FUNCTION_BLOCK FB_TriLogic (* Logique de tri - BLOCK seulement si couleur differente *)
  (* Standard: 61499-2 *)
  (* Version 2.0, 20/01/2026, Claude, Schneider Electric, Block seulement si changement de couleur *)
  PACKAGE Main;
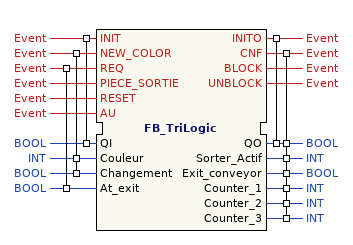
  EVENT_INPUT
    INIT WITH QI; (* Initialization Request *)
    NEW_COLOR WITH Couleur, Changement; (* Nouvelle couleur detectee *)
    REQ WITH At_exit; (* Cyclic update *)
    PIECE_SORTIE; (* Piece a quitte le systeme (front descendant At_exit) *)
    RESET; (* Reset compteurs *)
    AU; (* Arret urgence *)
  END_EVENT
  EVENT_OUTPUT
    INITO WITH QO; (* Initialization Confirm *)
    CNF WITH QO, Sorter_Actif, Exit_conveyor, Counter_1, Counter_2, Counter_3; (* Execution Confirmation *)
    BLOCK; (* Bloquer entree (couleur differente) *)
    UNBLOCK; (* Debloquer entree *)
  END_EVENT
  VAR_INPUT
    QI : BOOL; (* Input event qualifier *)
    Couleur : INT; (* 1=Bleu, 2=Vert, 3=Gris *)
    Changement : BOOL; (* TRUE si couleur differente *)
    At_exit : BOOL; (* Capteur sortie *)
  END_VAR
  VAR_OUTPUT
    QO : BOOL; (* Output event qualifier *)
    Sorter_Actif : INT; (* Sorter actif (1-3) *)
    Exit_conveyor : BOOL; (* Convoyeur sortie actif *)
    Counter_1 : INT; (* Compteur bleu *)
    Counter_2 : INT; (* Compteur vert *)
    Counter_3 : INT; (* Compteur gris *)
  END_VAR
  VAR
    Couleur_EnCours : INT; (* Couleur piece en cours de tri *)
    Couleur_Suivante : INT; (* Couleur piece suivante (si differente) *)
    Is_Blocked : BOOL; (* TRUE si entree bloquee *)
  END_VAR
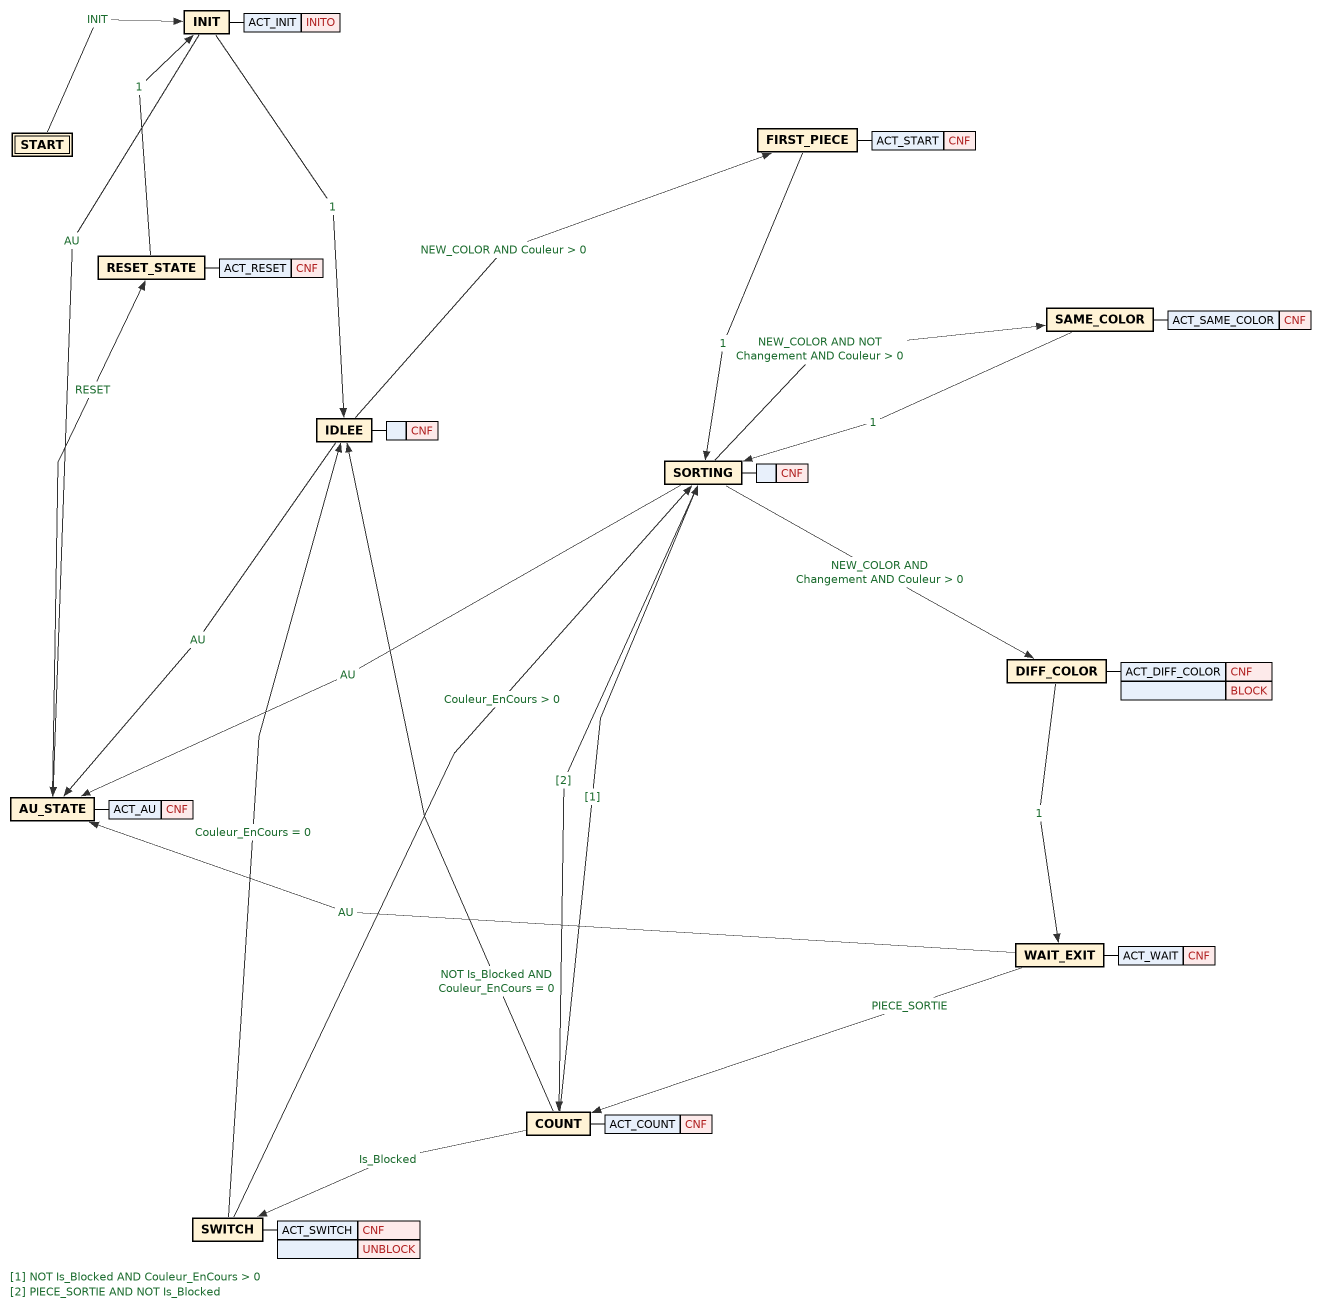
  EC_STATES
    START; (* Initial State *)
    INIT : ACT_INIT -> INITO; (* Initialization *)
    IDLEE : -> CNF; (* En attente - pas de piece *)
    FIRST_PIECE : ACT_START -> CNF; (* Premiere piece - activer sorter *)
    SORTING : -> CNF; (* Tri en cours *)
    SAME_COLOR : ACT_SAME_COLOR -> CNF; (* Meme couleur - pas de blocage *)
    DIFF_COLOR : ACT_DIFF_COLOR -> CNF, -> BLOCK; (* Couleur differente - BLOCK *)
    WAIT_EXIT : ACT_WAIT -> CNF; (* Attendre sortie piece *)
    COUNT : ACT_COUNT -> CNF; (* Piece sortie - compter *)
    SWITCH : ACT_SWITCH -> CNF, -> UNBLOCK; (* Changer sorter - UNBLOCK *)
    AU_STATE : ACT_AU -> CNF; (* Arret urgence *)
    RESET_STATE : ACT_RESET -> CNF; (* Reset *)
  END_STATES
  EC_TRANSITIONS
    START TO INIT := INIT;
    INIT TO IDLEE := 1;
    IDLEE TO FIRST_PIECE := NEW_COLOR AND Couleur > 0;
    FIRST_PIECE TO SORTING := 1;
    SORTING TO SAME_COLOR := NEW_COLOR AND NOT Changement AND Couleur > 0;
    SORTING TO DIFF_COLOR := NEW_COLOR AND Changement AND Couleur > 0;
    SAME_COLOR TO SORTING := 1;
    DIFF_COLOR TO WAIT_EXIT := 1;
    WAIT_EXIT TO COUNT := PIECE_SORTIE;
    SORTING TO COUNT := PIECE_SORTIE AND NOT Is_Blocked;
    COUNT TO SWITCH := Is_Blocked;
    COUNT TO SORTING := NOT Is_Blocked AND Couleur_EnCours > 0;
    COUNT TO IDLEE := NOT Is_Blocked AND Couleur_EnCours = 0;
    SWITCH TO SORTING := Couleur_EnCours > 0;
    SWITCH TO IDLEE := Couleur_EnCours = 0;
    IDLEE TO AU_STATE := AU;
    SORTING TO AU_STATE := AU;
    WAIT_EXIT TO AU_STATE := AU;
    AU_STATE TO RESET_STATE := RESET;
    RESET_STATE TO INIT := 1;
    INIT TO AU_STATE := AU;
  END_TRANSITIONS
  ALGORITHM ACT_INIT IN ST: (* Initialization *)
QO := TRUE;
Sorter_Actif := 0;
Exit_conveyor := FALSE;
Couleur_EnCours := 0;
Couleur_Suivante := 0;
Is_Blocked := FALSE;
Counter_1 := 0;
Counter_2 := 0;
Counter_3 := 0;
  END_ALGORITHM
  ALGORITHM ACT_START IN ST: (* Premiere piece - activer sorter *)
(* Premiere piece detectee - activer le sorter *)
Couleur_EnCours := Couleur;
Sorter_Actif := Couleur;
Exit_conveyor := TRUE;
Is_Blocked := FALSE;
  END_ALGORITHM
  ALGORITHM ACT_SAME_COLOR IN ST: (* Meme couleur - continuer sans bloquer *)
(* Meme couleur que precedente - pas de blocage *)
(* Le sorter est deja bon, on continue *)
Exit_conveyor := TRUE;
  END_ALGORITHM
  ALGORITHM ACT_DIFF_COLOR IN ST: (* Couleur differente - bloquer et memoriser *)
(* Couleur DIFFERENTE - bloquer l'entree et memoriser *)
Couleur_Suivante := Couleur;
Is_Blocked := TRUE;
(* IMPORTANT: garder le sorter actuel jusqu'a ce que la piece sorte *)
Exit_conveyor := TRUE;
  END_ALGORITHM
  ALGORITHM ACT_WAIT IN ST: (* Attendre sortie piece *)
(* Attendre que la piece en cours sorte *)
(* Garder le sorter actuel actif *)
Sorter_Actif := Couleur_EnCours;
Exit_conveyor := TRUE;
  END_ALGORITHM
  ALGORITHM ACT_COUNT IN ST: (* Compter la piece sortie *)
(* Piece sortie - incrementer compteur *)
IF Couleur_EnCours = 1 THEN
    Counter_1 := Counter_1 + 1;
ELSIF Couleur_EnCours = 2 THEN
    Counter_2 := Counter_2 + 1;
ELSIF Couleur_EnCours = 3 THEN
    Counter_3 := Counter_3 + 1;
END_IF;

(* Preparer pour la suite *)
IF Is_Blocked THEN
    (* On va changer de couleur *)
    Couleur_EnCours := Couleur_Suivante;
ELSE
    (* Pas de piece en attente - on garde la meme couleur active *)
    (* Couleur_EnCours reste inchange *)
   Couleur_EnCours := Couleur;
END_IF;
  END_ALGORITHM
  ALGORITHM ACT_SWITCH IN ST: (* Changer sorter et debloquer *)
(* Changer le sorter pour la nouvelle couleur *)
Sorter_Actif := Couleur_EnCours;
Couleur_Suivante := 0;
Is_Blocked := FALSE;
Exit_conveyor := TRUE;
  END_ALGORITHM
  ALGORITHM ACT_AU IN ST: (* Arret urgence *)
(* Tout arreter *)
Sorter_Actif := 0;
Exit_conveyor := FALSE;
Couleur_EnCours := 0;
Couleur_Suivante := 0;
Is_Blocked := FALSE;
  END_ALGORITHM
  ALGORITHM ACT_RESET IN ST: (* Reset complet *)
(* Reset compteurs et etats *)
QO := TRUE;
Sorter_Actif := 0;
Exit_conveyor := FALSE;
Couleur_EnCours := 0;
Couleur_Suivante := 0;
Is_Blocked := FALSE;
Counter_1 := 0;
Counter_2 := 0;
Counter_3 := 0;
  END_ALGORITHM
END_FUNCTION_BLOCK
